PROGRAM CountToExample
VAR
	// An array of jobs to do
	myWorker: MyWorker;
	counting: ARRAY[1..10] OF CountToJob := [(CountTo := 200, Worker := myWorker.Base)];
	i: UDINT;
	
	// Rising edge will trigger the state change.
	bStart: BOOL;
END_VAR

IF bStart THEN
	bStart := FALSE;
	FOR i := 1 TO 10 DO
	counting[i].Start();
	END_FOR	
	
END_IF

END_PROGRAM

(* stored: Version 1.1.0.1
   POU CountToExample: Id {5fde126a-5e43-4858-8366-2e235f667e4f}, SpecialFunc None *)
